// Mitsubishi GX Works2 project: wandEx02   PLC: Q02/Q02H

PROGRAM MAIN
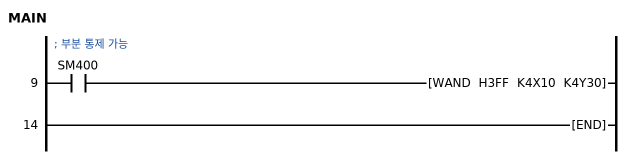
; 부분 통제 가능
9     LD      SM400
      WAND    H3FF K4X10 K4Y30
14    END
END_PROGRAM
